(* Schneider Machine Expert - Basic project A10 Descarga de Ar Silos, file version 2.7.0.0 *)
(* ProjectInformations: Name=Novo projeto *)

HARDWARE
  Cpu 0: TM221M16R/G
  EthernetConfiguration: NetworkName=M221, IpAllocationMode=FixedAddress, IpAddress=0.0.0.0, SubnetMask=0.0.0.0
  SerialLineConfiguration: Baud=Baud19200, Parity=ParityEven, DataBits=DataBits8, StopBits=StopBits1, PhysicalMedium=PhysicalMediumRs485, TransmissionMode=TransmissionModeModbusRtu, SlaveId=1, Addressing=SlaveAddressing
  MastTask: UsePeriodScanMode=false, PeriodScan=100
  FastTask: Period=255
  CpuBehavior: StartingMode=StartAsPreviousState, AutoSaveRamOnEeprom=true, WatchdogPeriod=250

SYMBOLS  (address, symbol, comment, settings)
  %M0         "Habilita Pulso Ar"
  %M1         "Descarga de Ar"
  %TM0        [Preset=5, Base=OneSecond]
  %I0.0       "Chave Desliga"
  %I0.1       "Chave liga Ar"
  %Q0.0       "Valvula Puls Ar"

POU Novo POU
  (* SectionNumber=1 *)

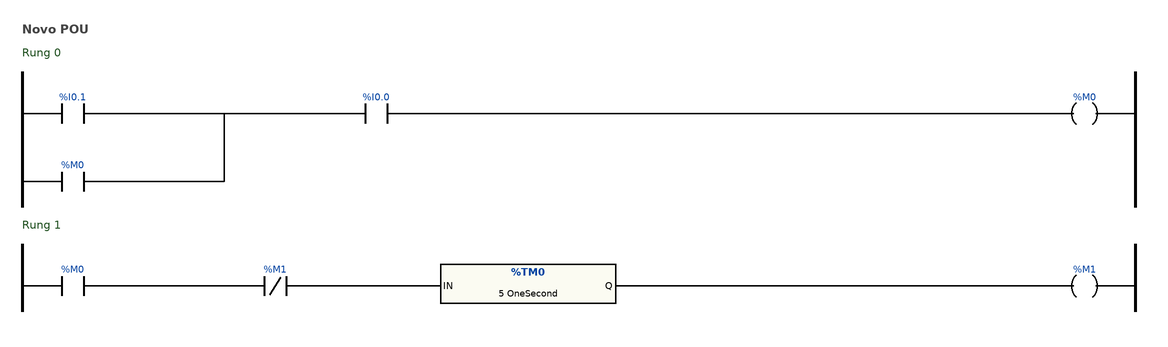

// Rung 0
  LD %I0.1
  OR %M0
  AND %I0.0
  ST %M0
  // as ST:
  //   %M0 := (%I0.1 OR %M0) AND %I0.0;

// Rung 1
  BLK %TM0
  LD %M0
  ANDN %M1
  IN
  OUT_BLK
  LD Q
  ST %M1
  END_BLK
  // as ST:
  //   %TM0(IN := %M0 AND NOT %M1);
  //   %M1 := %TM0.Q;
